{attribute addProperty BoxType "EK1100-0000-0018"}
{attribute addProperty Id "Beckhoff_EL3xxx_0030EK1122Beckhoff_EL3xxx_0030EK1122_A8C7E601162A_0001_EL3174_0030_0016EL3174_B7B5302521026.25A_0002_EL3314_0030_0021EL3314_AAA7BA7127434.25A_0003_EL3681_0030_0021EL3681_AB553B5016220.25A_0004_EL3201_0030_0022EL3201_73D65BA516320.375A_0005_EL3202_0030_0022EL3202_CEE8F25A24430.5A_0006_EL3356_0030_0025EL3356_AAE78EE214618.25A_0007_EL3692_0030_0021EL3692_4E8506B127434.25"}
{attribute addProperty CRC "755497836"}
{attribute addProperty SizeInBites "1489"}
{attribute addProperty SizeInBytes "186.125"}
TYPE Beckhoff_EL3xxx_0030_2D07FB6C EXTENDS EK1100_179A0949 :
STRUCT
	{attribute addProperty Name "Beckhoff_EL3xxx_0030EK1122"}
	Beckhoff_EL3xxx_0030EK1122 : Beckhoff_EL3xxx_0030EK1122_A8C7E601;
	{attribute addProperty Name "A_0001_EL3174_0030_0016"}
	A_0001_EL3174_0030_0016 : EL3174_B7B53025;
	{attribute addProperty Name "A_0002_EL3314_0030_0021"}
	A_0002_EL3314_0030_0021 : EL3314_AAA7BA71;
	{attribute addProperty Name "A_0003_EL3681_0030_0021"}
	A_0003_EL3681_0030_0021 : EL3681_AB553B50;
	{attribute addProperty Name "A_0004_EL3201_0030_0022"}
	A_0004_EL3201_0030_0022 : EL3201_73D65BA5;
	{attribute addProperty Name "A_0005_EL3202_0030_0022"}
	A_0005_EL3202_0030_0022 : EL3202_CEE8F25A;
	{attribute addProperty Name "A_0006_EL3356_0030_0025"}
	A_0006_EL3356_0030_0025 : EL3356_AAE78EE2;
	{attribute addProperty Name "A_0007_EL3692_0030_0021"}
	A_0007_EL3692_0030_0021 : EL3692_4E8506B1;
END_STRUCT
END_TYPE

(* stored: Version 1.2.0.0, ProductVersion 3.1.4024.9
   DUT Beckhoff_EL3xxx_0030_2D07FB6C: Id {67e72c66-fd7d-4869-b7a3-251280bbca2b} *)
